// TIA Portal V15.1 export
// export: Created 2022-12-20T09:13:23.8328509Z, ExportSetting None, DisplayName Totally Integrated Automation Portal, DisplayVersion V15.1 Update 1, DisplayName TIA Portal Openness, DisplayVersion V15.1, DisplayName SINAMICS Startdrive Advanced, DisplayVersion V15.1, DisplayName G130, G150, S120, S150, SINAMICS MV, S210, DisplayVersion V15.1, DisplayName G110M, G120, G120C, G120D, G120P, DisplayVersion V15.1, DisplayName STEP 7 Professional, DisplayVersion V15.1 Update 1, DisplayName STEP 7 Safety, DisplayVersion V15.1, DisplayName WinCC Professional, DisplayVersion V15.1 Update 1, DisplayName SIMATIC Visualization Architect, DisplayVersion V15.1
FUNCTION_BLOCK "PLC_ROBOT_FB"   // FB512, FBD
TITLE = PLC_ROBOT_FB
{ S7_Optimized_Access := 'TRUE' }
// Handle robot functions
// stored: AutoNumber false, MemoryReserve 100, SetENOAutomatically False
   VAR
      Robot_AO_BrakeTest { ExternalAccessible := 'False'; ExternalVisible := 'False'; ExternalWritable := 'False'} : "CM_Robot_AO_BrakeTest_FB";   // Robot add on block for brake test
   END_VAR
BEGIN

REGION Network 1: ***Robot braketest***
   // Collection of robot braketest functions
END_REGION

REGION Network 2: Call robot breaktest block settings
   // Set the time of the day of the week a robot brake test should be performed
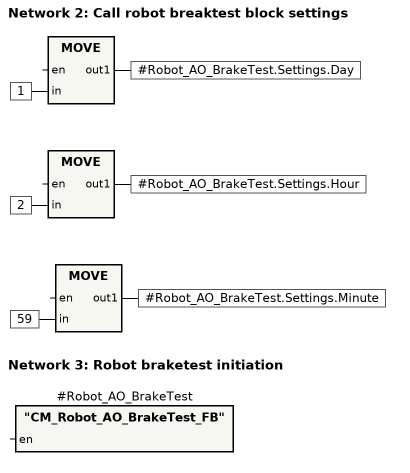
   #Robot_AO_BrakeTest.Settings.Day := 1;
   #Robot_AO_BrakeTest.Settings.Hour := 2;
   #Robot_AO_BrakeTest.Settings.Minute := 59;
END_REGION

REGION Network 3: Robot braketest initiation
   // Brake test of robots in the SA will be initiated on time or when a robot requests a brake test
   #Robot_AO_BrakeTest();   // "CM_Robot_AO_BrakeTest_FB"
END_REGION
END_FUNCTION_BLOCK
